// TIA Portal project "SPEEDGOAT_SimulaceSoustav_V20" (V20)

(* hardware
DEVICE "GSD device_1"  GSD.Device.PN
   slot 0: "Rack"  Rack  V1.0
   slot 0: "speedgoat-io750"  CIFX RE/PNS V3.4.19 - V3.4.x  1250.100  V3.4
      slot 0: "CIFX RE/PNS V3.4.19 - V3.4.x"  CIFX RE/PNS V3.4.19 - V3.4.x
      slot 1: "PN-IO"  PN-IO
         slot 1: "Port 1"  Port 1
         slot 2: "Port 2"  Port 2
   slot 1: "Model A - PN u"  4 Bytes Output
      slot 0: "4 Bytes Output"  4 Bytes Output
   slot 2: "Model A - PN y"  4 Bytes Input
      slot 0: "4 Bytes Input"  4 Bytes Input
DEVICE "S71500/ET200MP station_5"  S7-1500 station
   slot 0: "Rail_0"  Rack  6ES7 590-1***0-0AA0
   slot 1: "1500_ControlPLC"  CPU 1516-3 PN/DP  6ES7 516-3AN01-0AB0  V2.1
      slot 3: "CPU display_1"  6ES7591-1BA00-0AA0
   slot 2: "DI 32x24VDC HF_1"  DI 32x24VDC HF  6ES7 521-1BL00-0AB0  V2.0
   slot 3: "DQ 32x24VDC/0.5A HF_1"  DQ 32x24VDC/0.5A HF  6ES7 522-1BL01-0AB0  V1.0
   slot 4: "AQ 4xU/I ST_1"  AQ 4xU/I ST  6ES7 532-5HD00-0AB0  V2.0
   slot 5: "AI 8xU/I/RTD/TC ST_1"  AI 8xU/I/RTD/TC ST  6ES7 531-7KF00-0AB0  V2.0
DEVICE "GSD device_2"  GSD.Device.PN
   slot 0: "Rack"  Rack  V1.0
   slot 0: "speedgoat-io752"  CIFX RE/PNS V3.4.19 - V3.4.x  1250.100  V3.4
      slot 0: "CIFX RE/PNS V3.4.19 - V3.4.x"  CIFX RE/PNS V3.4.19 - V3.4.x
      slot 1: "PN-IO"  PN-IO
         slot 1: "Port 1"  Port 1
         slot 2: "Port 2"  Port 2
   slot 1: "Model C - PN u"  4 Bytes Output
      slot 0: "4 Bytes Output"  4 Bytes Output
   slot 2: "Model C - PN y"  4 Bytes Input
      slot 0: "4 Bytes Input"  4 Bytes Input
DEVICE "GSD device_3"  GSD.Device.PN
   slot 0: "Rack"  Rack  V1.0
   slot 0: "speedgoat-io751"  CIFX RE/PNS V3.4.19 - V3.4.x  1250.100  V3.4
      slot 0: "CIFX RE/PNS V3.4.19 - V3.4.x"  CIFX RE/PNS V3.4.19 - V3.4.x
      slot 1: "PN-IO"  PN-IO
         slot 1: "Port 1"  Port 1
         slot 2: "Port 2"  Port 2
   slot 1: "Model B - PN u"  4 Bytes Output
      slot 0: "4 Bytes Output"  4 Bytes Output
   slot 2: "Model B - PN y"  4 Bytes Input
      slot 0: "4 Bytes Input"  4 Bytes Input
DEVICE "HMI_1"  KTP900 Basic PN
   slot 0: "HMI_1"  KTP900 Basic PN  6AV2 123-2JB03-0AX0  15.1.0.0
   slot 1: "HMI_RT_1"  KTP900 Basic PN  6AV2 123-2JB03-0AX0  15.1.0.0
   slot 5: "HMI_1.IE_CP_1"  PROFINET Interface  15.0.1.0
      slot 1: "PROFINET Interface_1"  PROFINET Interface
         slot 1: "Port_1"  Port
DEVICE "GSD device_4"  GSD.Device.PN
   slot 0: "Rack"  Rack  V1.0
   slot 0: "speedgoat-io752_1"  CIFX RE/PNS V3.4.19 - V3.4.x  1250.100  V3.4
      slot 0: "CIFX RE/PNS V3.4.19 - V3.4.x"  CIFX RE/PNS V3.4.19 - V3.4.x
      slot 1: "PN-IO"  PN-IO
         slot 1: "Port 1"  Port 1
         slot 2: "Port 2"  Port 2
   slot 1: "Model C - PN u"  4 Bytes Output
      slot 0: "4 Bytes Output"  4 Bytes Output
   slot 2: "Model C - PN y"  4 Bytes Input
      slot 0: "4 Bytes Input"  4 Bytes Input
*)

// ===== PLC "1500_ControlPLC"  CPU 1516-3 PN/DP =====

VAR_GLOBAL   // PLC tag table "Process"
   "Only_Model_A_PN" AT %M20.0 : Bool;
   "Only_Model_B_PN" AT %M20.1 : Bool;
   "Only_Model_C_PN" AT %M20.2 : Bool;
   "SetPoint A" AT %MD54 : Real;
   "SetPoint B" AT %MD58 : Real;
   "SetPoint C" AT %MD62 : Real;
   "Model A - Reset" AT %M20.4 : Bool;
   "Model B - Reset" AT %M20.5 : Bool;
   "Model C - Reset" AT %M20.6 : Bool;
   "Connection_LOOPBACK" AT %M20.7 : Bool;   // Activates copying PROFINET input to output
   "Model A - PN u" AT %QD30 : Real;   // System A input (u) via PROFINET
   "Model B - PN u" AT %QD34 : Real;   // System B input (u) via PROFINET
   "Model C - PN u" AT %QD38 : Real;   // System C input (u) via PROFINET
   "Model A - PN y" AT %ID0 : Real;   // System A output (y) via PROFINET
   "Model B - PN y" AT %ID4 : Real;   // System B output (y) via PROFINET
   "Model C - PN y" AT %ID8 : Real;   // System C output (y) via PROFINET
   "Connection_PROFINET" AT %M20.3 : Bool;   // Activates closed loop control via PROFINET
   "Connection_LOCALMODEL" AT %M21.0 : Bool;   // Activates closed loop control with LOCAL MODELS
   "MEM 1" AT %M200.0 : Bool;   // E
   "MEM 2" AT %M200.1 : Bool;   // E
   "MEM 3" AT %M200.2 : Bool;   // E
   "MEM 4" AT %M200.3 : Bool;   // E
   "MEM 5" AT %M200.4 : Bool;   // E
   "MEM 6" AT %M200.5 : Bool;
   "MEM 7" AT %M200.6 : Bool;
   "MEM 8" AT %M200.7 : Bool;
   "MEM 9" AT %M201.0 : Bool;
   "MEM 10" AT %M201.1 : Bool;
   "MEM 11" AT %M201.2 : Bool;
   "MEM 12" AT %M201.3 : Bool;
   "MEM 13" AT %M201.4 : Bool;
   "MEM 14" AT %M201.5 : Bool;
   "MEM 15" AT %M201.6 : Bool;
   "MEM 16" AT %M201.7 : Bool;
   "MEM 17" AT %M202.0 : Bool;
   "MEM 18" AT %M202.1 : Bool;
   "Connection_NOCONNECTION" AT %M21.1 : Bool;
   "Connection_MANUALVALUE" AT %M21.2 : Bool;
   "resetModels" AT %M21.3 : Bool;
   "SetPoint D" AT %MD66 : Real;
   "Model D - PN u" AT %QD42 : Real;   // System D input (u) via PROFINET
   "Model D - PN y" AT %ID32 : Real;   // System D output (y) via PROFINET
   "EnablePID_D" AT %M21.4 : Bool;
   "SP DEMO" AT %M21.5 : Bool;
   "SP BINVAL" AT %M21.6 : Bool;
END_VAR

DATA_BLOCK "LSim_PDT1_DB"   // DB1
{ S7_Optimized_Access := 'TRUE' }
VERSION : 2.01
// stored: InstanceOfName LSim_PDT1
"LSim_PDT1"
BEGIN
END_DATA_BLOCK

DATA_BLOCK "Model_Params"   // DB2
{ S7_Optimized_Access := 'TRUE' }
VERSION : 0.1
   VAR
      "Model A" : Struct
         tmLag1 : Real := 3.0;
         tmLag2 : Real := 0.3;
         gain : Real := 1.25;
         cycle : Real := 0.2;
         maxOut : Real := 100.0;
         minOut : Real := 0.0;
      END_STRUCT;
      "Model B" : Struct
         tmLag1 : Real := 1.2;
         tmLag2 : Real := 0.25;
         gain : Real := 1.45;
         cycle : Real := 0.1;
         maxOut : Real := 100.0;
         minOut : Real := 0.0;
      END_STRUCT;
      "Model C" : Struct
         omega : Real := 2.0;
         damp : Real := 0.2;
         gain : Real := 1.33;
         cycle : Real := 0.05;
         maxOut : Real := 100.0;
         minOut : Real := 0.0;
      END_STRUCT;
   END_VAR
BEGIN
END_DATA_BLOCK

DATA_BLOCK "LSim_PT2aper_DB"   // DB3
{ S7_Optimized_Access := 'TRUE' }
VERSION : 2.01
// stored: InstanceOfName LSim_PT2aper
"LSim_PT2aper"
BEGIN
END_DATA_BLOCK

DATA_BLOCK "LSim_PT2osc_DB"   // DB8
{ S7_Optimized_Access := 'TRUE' }
VERSION : 2.01
// stored: InstanceOfName LSim_PT2osc
"LSim_PT2osc"
BEGIN
END_DATA_BLOCK

FUNCTION_BLOCK "LSim_PT2osc"   // FB52, SCL
{ S7_Optimized_Access := 'TRUE' }
VERSION : 2.01
   VAR_INPUT
      calcParam : Bool;   // recalculate with new parameters
      input : Real;   // input signal
      omega : Real := 2.0;   // angular frequency of the undampened vibrations [1/sec]
      damp : Real := 0.2;   // damping (0 < D < 1)
      gain : Real := 1.0;   // gain factor
      cycle : Real := 0.1;   // cyclic time [sec]
      maxOut : Real := 100.0;   // max. output limit
      minOut : Real;   // min. output limit
      reset : Bool;   // resets all relevant parameters to ‘0’ including the output
   END_VAR
   VAR_OUTPUT
      error : Bool;   // error (0 >= damp >= 1 or #omega <= 0)
      status : Word;   // status (if #error = TRUE then status = 16#8001)
      maxReached : Bool;   // output has reached max. limit
      minReached : Bool;   // output has reached min. limit
      output : Real;   // output signal (if #error = FALSE)
   END_VAR
   VAR
      statRxn2 : Real;   // delayed input signal (n-2)
      statRxn1 : Real;   // delayed input signal (n-1)
      statRyn2 : Real;   // delayed output signal (n-2)
      statRyn1 : Real;   // delayed output signal (n-1)
      statRb1 : Real;
      statRb2 : Real;
      statRa1 : Real;
      statRa2 : Real;
      statRo : Real;
      statSigma : Real;
      statNue : Real;
      statOverfirst : Bool;
      statOutput : Real;
   END_VAR
BEGIN
   //=============================================================================
   //SIEMENS AG
   //(c)Copyright 2017 All Rights Reserved
   //-----------------------------------------------------------------------------
   //Library:       Library for Controlled System Simulation
   //Tested with:   S7-1500 FW V2.0 / S7-1200 FW V4.2
   //Engineering:   STEP 7 V14 Upd2 (TIA Portal)
   //Restrictions:  Cyclic interrupt
   //Requirements:  memory card needed for S7-1500
   //Functionality: Simulation of a vibrating PT2-System
   //
   //                  gain
   //  F(p) = ----------------------------------
   //         SQR(p/omega) + 2*damp*p/omega + 1
   //          
   //  Call the simulation in a cyclic interrupt with
   //  cyclic interrupt time at least = tmLag1/10!
   //-----------------------------------------------------------------------------
   //Change log table:
   //Version  Date       Expert in charge                Changes applied
   //02.00.00 03.02.2016 Siemens Industry Online Support Release (STEP 7 V13 SP1)
   //02.00.01 02.03.2017 Siemens Industry Online Support Release (STEP 7 V14)
   //=============================================================================

   // check parameter
   IF #damp >= 1 OR #damp <= 0 OR #omega <= 0 THEN
     #error := TRUE;
     #status := W#16#8001;
     #statRxn1 := 0.0;
     #statRyn1 := 0.0;
     #statRxn2 := 0.0;
     #statRyn2 := 0.0;
     #statOutput := 0;
     #output := 0;
     RETURN;
   ELSE
     #error := FALSE;
     #status := W#16#0000;     // no error 
   END_IF;

   // calculates the z-parameter for the difference equatation
   IF #calcParam = True THEN
   // Calculate z-parameters for oscillating PT2-System
   #statRo := EXP(-2*#omega*#damp*#cycle);
   #statSigma := (COS(#omega * #cycle * SQRT(1 - SQR(#damp)))) * EXP(-#damp*#omega*#cycle);
   #statNue := (SIN(#omega*#cycle*SQRT(1-SQR(#damp)))) * (EXP(-#damp*#omega*#cycle)) * (#damp / SQRT(1 - SQR(#damp)));
   #statRa1 := -2*#statSigma;
   #statRa2 := #statRo;
   #statRb1 := #gain*(1 - #statSigma - #statNue);
   #statRb2 := #gain*(#statRo - #statSigma + #statNue);
   END_IF;

   // reset Memory
   IF #reset = True THEN
     #statRxn1 := 0.0;
     #statRyn1 := 0.0;
     #statRxn2 := 0.0;
     #statRyn2 := 0.0;
     #statOutput:=0;
     #error := False;
     #status := W#16#0000;
   END_IF;

   // save delayed output signals
   #statRyn2:=#statRyn1;
   #statRyn1:= #statOutput;

   // difference equatation for PT2-System
   #statOutput := #statRxn1* #statRb1 + #statRxn2*#statRb2 - #statRyn1*#statRa1 - #statRyn2*#statRa2;

   // save delayed input signals
   #statRxn2 := #statRxn1;
   #statRxn1 := #input;

   // max limit of acutating variable
   IF #statOutput > #maxOut THEN
     #statOutput := #maxOut;
     #maxReached:= True;
   ELSE
     #maxReached := False;
   END_IF;

   // min limit of acutating variable
   IF #statOutput < #minOut THEN
     #statOutput := #minOut;
     #minReached := True;
   ELSE
     #minReached := False;
   END_IF;

   #output := #statOutput;
END_FUNCTION_BLOCK

FUNCTION_BLOCK "LSim_PT2aper"   // FB53, SCL
{ S7_Optimized_Access := 'TRUE' }
VERSION : 2.01
   VAR_INPUT
      calcParam : Bool;   // recalculate with new parameters
      input : Real;   // input signal
      tmLag1 : Real := 2.0;   // time constant T1 [sec]
      tmLag2 : Real := 0.2;   // time constant T2 [sec]
      gain : Real := 1.0;   // gain factor
      cycle : Real := 0.1;   // cyclic time [sec]
      maxOut : Real := 100.0;   // max. output limit
      minOut : Real;   // min. output limit
      reset : Bool;   // resets all relevant parameters to ‘0’ including the output
   END_VAR
   VAR_OUTPUT
      error : Bool;   // error (#tmLag1 <= 0 or #tmLag2 <= 0 or #tmLag1 = #tmLag2)
      status : Word;   // status (if #error = TRUE then status = 16#8001)
      maxReached : Bool;   // output has reached max. limit
      minReached : Bool;   // output has reached min. limit
      output : Real;   // output signal (if #error = FALSE)
   END_VAR
   VAR
      statRxn2 : Real;   // delayed input signal (n-2)
      statRxn1 : Real;   // delayed input signal (n-1)
      statRyn2 : Real;   // delayed output signal (n-2)
      statRyn1 : Real;   // delayed output signal (n-1)
      statRf1 : Real;
      statRf2 : Real;
      statRe1 : Real;
      statRe2 : Real;
      statAlpha : Real;
      statBeta : Real;
      statGamma : Real;
      statDelta : Real;
      statOverfirst : Bool;
      statOutput : Real;   // Output signal
   END_VAR
BEGIN
   //=============================================================================
   //SIEMENS AG
   //(c)Copyright 2017 All Rights Reserved
   //-----------------------------------------------------------------------------
   //Library:       Library for Controlled System Simulation
   //Tested with:   S7-1500 FW V2.0 / S7-1200 FW V4.2
   //Engineering:   STEP 7 V14 Upd2 (TIA Portal)
   //Restrictions:  Cyclic interrupt
   //Requirements:  memory card needed for S7-1500
   //Functionality: Simulation of a aperiodic PT2-System
   //  
   //                    gain
   //  F(p) = -----------------------------
   //         (tmLag1*p + 1)*(tmLag2*p + 1)
   //         
   //  Call the simulation in a cyclic interrupt with
   //  cyclic interrupt time at least = tmLag1/10!
   //-----------------------------------------------------------------------------
   //Change log table:
   //Version  Date       Expert in charge                Changes applied
   //02.00.00 03.02.2016 Siemens Industry Online Support Release (STEP 7 V13 SP1)
   //02.00.01 02.03.2017 Siemens Industry Online Support Release (STEP 7 V14)
   //=============================================================================

   // check parameter
   IF #tmLag1 <= 0 OR #tmLag2 <= 0 OR #tmLag1 = #tmLag2 THEN
     #error := TRUE;
     #status := W#16#8001;     // Parameter Error
     #statRxn1 := 0.0;
     #statRyn1 := 0.0;
     #statRxn2 := 0.0;
     #statRyn2 := 0.0;
     #statOutput := 0;
     #output := 0;
     RETURN;
   ELSE
     #error := FALSE;
     #status := W#16#0000;     // no error
   END_IF;

   // calculates the z-parameter for the difference equatation
   IF #calcParam = True OR NOT #statOverfirst THEN
     #statOverfirst := 1;
     // Calculate z-parameters for IT1-System
     #statAlpha := EXP(- #cycle / #tmLag1);
     #statBeta := EXP(- #cycle / #tmLag2);
     #statGamma := #tmLag1 / (#tmLag1 - #tmLag2);
     #statDelta := #tmLag2 / (#tmLag1 - #tmLag2);
     #statRe1 := - #statAlpha - #statBeta;
     #statRe2 := #statAlpha * #statBeta;
     #statRf1 := #gain * (1 - #statGamma * #statAlpha + #statDelta * #statBeta);
     #statRf2 := #gain * (#statAlpha * #statBeta - #statGamma * #statBeta + #statAlpha * #statDelta);
   END_IF;

   // reset Memory
   IF #reset = True THEN
     #statRxn1 := 0.0;
     #statRyn1 := 0.0;
     #statRxn2 := 0.0;
     #statRyn2 := 0.0;
     #statOutput := 0;
   END_IF;
   //save delayed input signals
   #statRxn2 := #statRxn1;
   #statRxn1 := #input;

   //save delayed output signals
   #statRyn2:=#statRyn1;
   #statRyn1:= #statOutput;

   // difference equatation of the PT2-System
   #statOutput := #statRxn1* #statRf1 + #statRxn2*#statRf2 - #statRyn1*#statRe1 - #statRyn2*#statRe2;

   // max limit of acutating variable
   IF #statOutput > #maxOut THEN
     #statOutput := #maxOut;
     #maxReached:= True;
   ELSE
     #maxReached := False;
   END_IF;

   // min limit of acutating variable
   IF #statOutput < #minOut THEN
     #statOutput := #minOut;
     #minReached := True;
   ELSE
     #minReached := False;
   END_IF;

   #output := #statOutput;
END_FUNCTION_BLOCK

FUNCTION_BLOCK "LSim_PDT1"   // FB55, SCL
{ S7_Optimized_Access := 'TRUE' }
VERSION : 2.01
   VAR_INPUT
      calcParam : Bool;   // recalculate with new parameters
      input : Real;   // input signal
      tmLag1 : Real := 2.0;   // time constant T1 [sec]
      tmLag2 : Real := 0.2;   // time constant T2 [sec]
      gain : Real := 1.0;   // gain factor
      cycle : Real := 0.1;   // cyclic time [sec]
      maxOut : Real := 100.0;   // max. output limit
      minOut : Real;   // min. output limit
      reset : Bool;   // resets all relevant parameters to ‘0’ including the output
   END_VAR
   VAR_OUTPUT
      error : Bool;   // error (#tmLag1 <= 0 or #tmLag2 <= 0)
      status : Word;   // status (if #error = TRUE then status = 16#8001)
      maxReached : Bool;   // output has reached max. limit
      minReached : Bool;   // output has reached min. limit
      output : Real;   // output signal (if #error = FALSE)
   END_VAR
   VAR
      statRxn2 : Real;   // delayed input signal (n-2)
      statRxn1 : Real;   // delayed input signal (n-1)
      statRyn2 : Real;   // delayed output signal (n-2)
      statRyn1 : Real;   // delayed output signal (n-1)
      statRb1 : Real;
      statRb0 : Real;
      statRa1 : Real;
      statOverfirst : Bool;
      statOutput : Real;
   END_VAR
BEGIN
   //=============================================================================
   //SIEMENS AG
   //(c)Copyright 2017 All Rights Reserved
   //-----------------------------------------------------------------------------
   //Library:       Library for Controlled System Simulation
   //Tested with:   S7-1500 FW V2.0 / S7-1200 FW V4.2
   //Engineering:   STEP 7 V14 Upd2 (TIA Portal)
   //Restrictions:  Cyclic interrupt
   //Requirements:  memory card needed for S7-1500
   //Functionality: Simulation of an PD-T1 System
   //
   //         gain * (1 + tmLag2*p)
   //  F(p) = ------------------------------
   //            (1 + tmLag1*p)
   //          
   //  Call the simulation in a cyclic interrupt with
   //  cyclic interrupt time at least = tmLag1/10!
   //-----------------------------------------------------------------------------
   //Change log table:
   //Version  Date       Expert in charge                Changes applied
   //02.00.00 03.02.2016 Siemens Industry Online Support Release (STEP 7 V13 SP1)
   //02.00.01 02.03.2017 Siemens Industry Online Support Release (STEP 7 V14)
   //=============================================================================

   // check parameter
   IF #tmLag1 <= 0 OR #tmLag2 <= 0 THEN
     #error := True;
     #status := W#16#8001;     // Parameter Error
     #statRxn1 := 0.0;
     #statRyn1 := 0.0;
     #statRxn2 := 0.0;
     #statRyn2 := 0.0;
     #statOutput := 0;
     #output := 0;
     RETURN;
   ELSE
     #error := FALSE;
     #status := W#16#0000;     // no error
   END_IF;

   // calculates the z-parameter for the difference equatation
   IF #calcParam = True OR NOT #statOverfirst THEN
     #statOverfirst := 1;
   // Calculate z-parameters for oscilating PT2-System
   #statRa1 := -EXP(-#cycle/#tmLag1);
   #statRb0 := #gain *(#tmLag2/#tmLag1);
   #statRb1 := #gain *(1 + #statRa1 - (#tmLag2/#tmLag1));
   END_IF;

   // reset Memory
   IF #reset = True THEN
     #statRxn1 := 0.0;
     #statRyn1 := 0.0;
     #statRxn2 := 0.0;
     #statRyn2 := 0.0;
     #statOutput:=0;
     #error := False;
     #status := W#16#0000;
   END_IF;

   // save delayed output-signals
   #statRyn1:= #statOutput;

   // difference equatation for PT2-system
   #statOutput := #input * #statRb0 +  #statRxn1* #statRb1 - #statRyn1*#statRa1;

   // save delayed input-signals
   #statRxn1 := #input;

   // max limit of acutating variable
   IF #statOutput > #maxOut THEN
     #statOutput := #maxOut;
     #maxReached:= True;
   ELSE
     #maxReached := False;
   END_IF;

   // min limit of acutating variable
   IF #statOutput < #minOut THEN
     #statOutput := #minOut;
     #minReached := True;
   ELSE
     #minReached := False;
   END_IF;

   #output := #statOutput;
END_FUNCTION_BLOCK

FUNCTION "ConnectionSwitch" : Void   // FC1, SCL
{ S7_Optimized_Access := 'TRUE' }
VERSION : 0.1
   VAR CONSTANT
      "Default value" : Real := 0.0;
   END_VAR
BEGIN
   IF "Connection_LOCALMODEL" THEN
       // Model A from local instance
       "PID_Compact_Control_A".Input := "LSim_PDT1_DB".output;
       "LSim_PDT1_DB".input := "PID_Compact_Control_A".Output;
       // Model B from local instance
       "PID_Compact_Control_B".Input := "LSim_PT2aper_DB".output;
       "LSim_PT2aper_DB".input := "PID_Compact_Control_B".Output;
       // Model C from local instance
       "PID_Compact_Control_C".Input := "LSim_PT2osc_DB".output;
       "LSim_PT2osc_DB".input := "PID_Compact_Control_C".Output;
       // Model D - nothing
       IF "EnablePID_D" = TRUE THEN
           "EnablePID_D" := FALSE;
       END_IF;

   ELSIF "Connection_PROFINET" THEN
       "EnablePID_D" := TRUE;
       // Model A from PN
       "PID_Compact_Control_A".Input := "Model A - PN y";
       "Model A - PN u" := "PID_Compact_Control_A".Output;
       // Model B from PN
       "PID_Compact_Control_B".Input := "Model B - PN y";
       "Model B - PN u" := "PID_Compact_Control_B".Output;
       // Model C from PN
       "PID_Compact_Control_C".Input := "Model C - PN y";
       "Model C - PN u" := "PID_Compact_Control_C".Output;
       // Model D fron PN
       "PID_Compact_Control_D".Input := "Model D - PN y";
       "Model D - PN u" := "PID_Compact_Control_D".Output;
   ELSIF "Connection_LOOPBACK" THEN
       "Model A - PN u" := "Model A - PN y";
       "Model B - PN u" := "Model B - PN y";
       "Model C - PN u" := "Model C - PN y";
       "Model D - PN u" := "Model D - PN y";
   ELSIF "Connection_MANUALVALUE" THEN
       "Model A - PN u" := "SetPoint A";
       "Model B - PN u" := "SetPoint B";
       "Model C - PN u" := "SetPoint C";
       "Model D - PN u" := "SetPoint D";
       IF "EnablePID_D" = TRUE THEN
           "EnablePID_D" := FALSE;
       END_IF;
   ELSE
       "Model A - PN u" := #"Default value";
       "Model B - PN u" := #"Default value";
       "Model C - PN u" := #"Default value";
       "Model D - PN u" := #"Default value";
       IF "EnablePID_D" = TRUE THEN
           "EnablePID_D" := FALSE;
       END_IF;
   END_IF;
END_FUNCTION

ORGANIZATION_BLOCK "Main"   // OB1, LAD, ProgramCycle
TITLE = "Main Program Sweep (Cycle)"
{ S7_Optimized_Access := 'TRUE' }
VERSION : 0.1
   VAR_INPUT
      Initial_Call : Bool;   // Initial call of this OB
      Remanence : Bool;   // =True, if remanent data are available
   END_VAR
   VAR_TEMP   // added for the SCL form of the ladder/FBD networks
      _w1 : Bool;
      _w2 : Bool;
      _w3 : Bool;
      _w4 : Bool;
      _w5 : Bool;
      _w6 : Bool;
   END_VAR
BEGIN

REGION Network 1: Connection switch
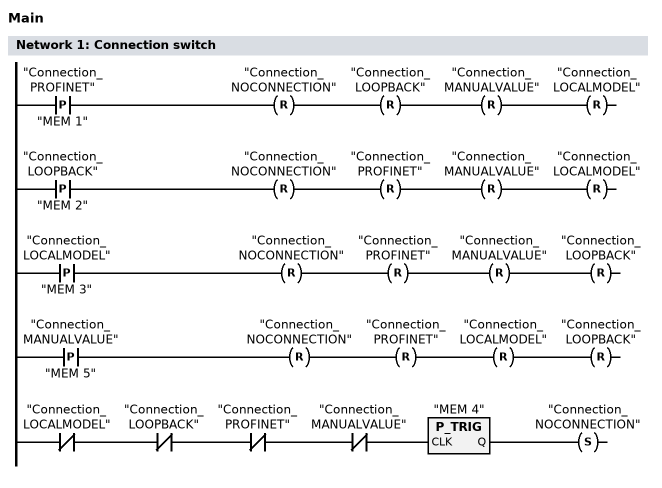
   RUNG wire#powerrail
      P_Contact(operand := "Connection_PROFINET", bit := "MEM 1")
      R_Coil( "Connection_NOCONNECTION" )
      R_Coil( "Connection_LOOPBACK" )
      R_Coil( "Connection_MANUALVALUE" )
      R_Coil( "Connection_LOCALMODEL" )
   END_RUNG
   RUNG wire#powerrail
      P_Contact(operand := "Connection_LOOPBACK", bit := "MEM 2")
      R_Coil( "Connection_NOCONNECTION" )
      R_Coil( "Connection_PROFINET" )
      R_Coil( "Connection_MANUALVALUE" )
      R_Coil( "Connection_LOCALMODEL" )
   END_RUNG
   RUNG wire#powerrail
      P_Contact(operand := "Connection_LOCALMODEL", bit := "MEM 3")
      R_Coil( "Connection_NOCONNECTION" )
      R_Coil( "Connection_PROFINET" )
      R_Coil( "Connection_MANUALVALUE" )
      R_Coil( "Connection_LOOPBACK" )
   END_RUNG
   RUNG wire#powerrail
      P_Contact(operand := "Connection_MANUALVALUE", bit := "MEM 5")
      R_Coil( "Connection_NOCONNECTION" )
      R_Coil( "Connection_PROFINET" )
      R_Coil( "Connection_LOCALMODEL" )
      R_Coil( "Connection_LOOPBACK" )
   END_RUNG
   RUNG wire#powerrail
      I_Contact( "Connection_LOCALMODEL" )
      I_Contact( "Connection_LOOPBACK" )
      I_Contact( "Connection_PROFINET" )
      I_Contact( "Connection_MANUALVALUE" )
      P_Trig( "MEM 4" )
      S_Coil( "Connection_NOCONNECTION" )
   END_RUNG
   // the same network as SCL:
   #_w1 := "Connection_PROFINET" AND NOT "MEM 1";   // rising edge of "Connection_PROFINET"
   "MEM 1" := "Connection_PROFINET";
   IF #_w1 THEN
       "Connection_NOCONNECTION" := FALSE;
       "Connection_LOOPBACK" := FALSE;
       "Connection_MANUALVALUE" := FALSE;
       "Connection_LOCALMODEL" := FALSE;
   END_IF;
   #_w2 := "Connection_LOOPBACK" AND NOT "MEM 2";   // rising edge of "Connection_LOOPBACK"
   "MEM 2" := "Connection_LOOPBACK";
   IF #_w2 THEN
       "Connection_NOCONNECTION" := FALSE;
       "Connection_PROFINET" := FALSE;
       "Connection_MANUALVALUE" := FALSE;
       "Connection_LOCALMODEL" := FALSE;
   END_IF;
   #_w3 := "Connection_LOCALMODEL" AND NOT "MEM 3";   // rising edge of "Connection_LOCALMODEL"
   "MEM 3" := "Connection_LOCALMODEL";
   IF #_w3 THEN
       "Connection_NOCONNECTION" := FALSE;
       "Connection_PROFINET" := FALSE;
       "Connection_MANUALVALUE" := FALSE;
       "Connection_LOOPBACK" := FALSE;
   END_IF;
   #_w4 := "Connection_MANUALVALUE" AND NOT "MEM 5";   // rising edge of "Connection_MANUALVALUE"
   "MEM 5" := "Connection_MANUALVALUE";
   IF #_w4 THEN
       "Connection_NOCONNECTION" := FALSE;
       "Connection_PROFINET" := FALSE;
       "Connection_LOCALMODEL" := FALSE;
       "Connection_LOOPBACK" := FALSE;
   END_IF;
   #_w5 := NOT "Connection_LOCALMODEL" AND NOT "Connection_LOOPBACK" AND NOT "Connection_PROFINET" AND NOT "Connection_MANUALVALUE";
   #_w6 := #_w5 AND NOT "MEM 4";   // rising edge
   "MEM 4" := #_w5;
   IF #_w6 THEN "Connection_NOCONNECTION" := TRUE; END_IF;
END_REGION
END_ORGANIZATION_BLOCK

ORGANIZATION_BLOCK "Control A"   // OB30, LAD, CyclicInterrupt
TITLE = Simulation and control of an PD-T1 System
{ S7_Optimized_Access := 'TRUE' }
VERSION : 0.1
   VAR_INPUT
      Initial_Call : Bool;   // Initial call of this OB
      Event_Count : Int;   // Events discarded
   END_VAR
BEGIN

REGION Network 1: Model of PDT1
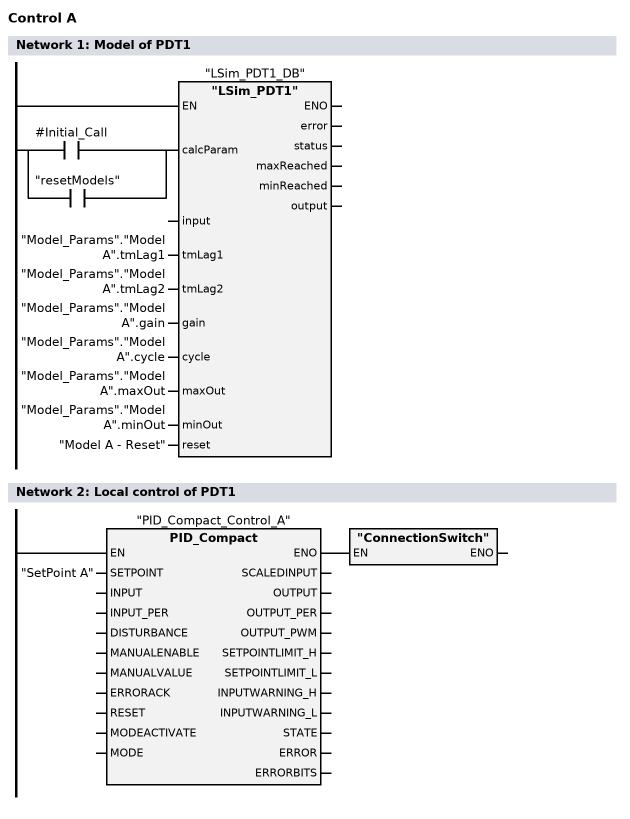
   RUNG wire#powerrail
      "LSim_PDT1_DB"(calcParam := wire#w1, input :=, tmLag1 := "Model_Params"."Model A".tmLag1, tmLag2 := "Model_Params"."Model A".tmLag2, gain := "Model_Params"."Model A".gain, cycle := "Model_Params"."Model A".cycle, maxOut := "Model_Params"."Model A".maxOut, minOut := "Model_Params"."Model A".minOut, reset := "Model A - Reset", error =>, status =>, maxReached =>, minReached =>, output =>)
   END_RUNG
   RUNG wire#powerrail
      Contact( #Initial_Call )
   END_RUNG wire#w1
   RUNG wire#powerrail
      Contact( "resetModels" )
   END_RUNG wire#w1
   // the same network as SCL:
   "LSim_PDT1_DB"(calcParam := #Initial_Call OR "resetModels",   // "LSim_PDT1"
                  tmLag1 := "Model_Params"."Model A".tmLag1,
                  tmLag2 := "Model_Params"."Model A".tmLag2,
                  gain := "Model_Params"."Model A".gain,
                  cycle := "Model_Params"."Model A".cycle,
                  maxOut := "Model_Params"."Model A".maxOut,
                  minOut := "Model_Params"."Model A".minOut,
                  reset := "Model A - Reset");
END_REGION

REGION Network 2: Local control of PDT1
   // ENO of a box is taken as its EN; it also drops when the box reports an error
   "PID_Compact_Control_A"(Setpoint := "SetPoint A");   // PID_Compact
   "ConnectionSwitch"();
END_REGION

REGION Network 3: Connection switch
END_REGION
END_ORGANIZATION_BLOCK

ORGANIZATION_BLOCK "Control B"   // OB31, LAD, CyclicInterrupt
TITLE = Simulation and control of an PT2aper system
{ S7_Optimized_Access := 'TRUE' }
VERSION : 0.1
   VAR_INPUT
      Initial_Call : Bool;   // Initial call of this OB
      Event_Count : Int;   // Events discarded
   END_VAR
BEGIN

REGION Network 1: Model of PT2aper
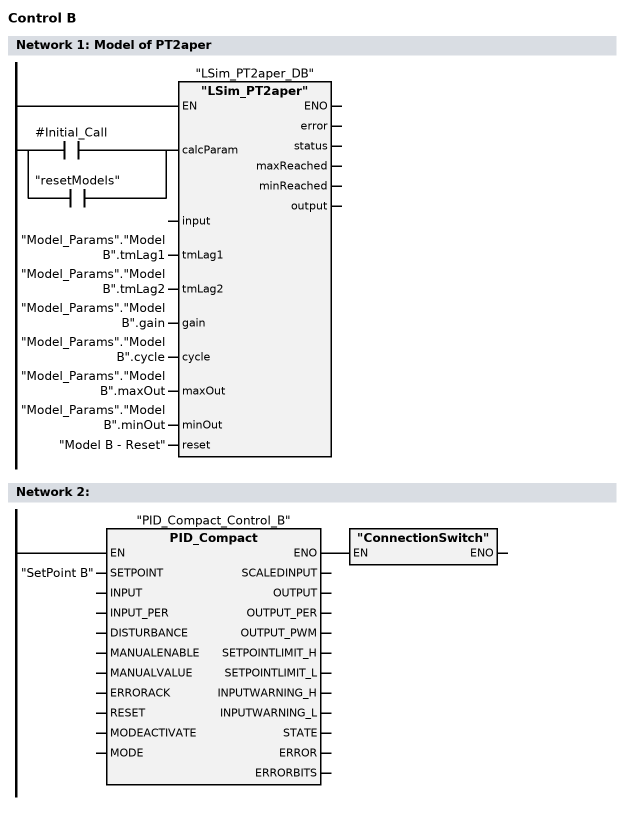
   RUNG wire#powerrail
      "LSim_PT2aper_DB"(calcParam := wire#w1, input :=, tmLag1 := "Model_Params"."Model B".tmLag1, tmLag2 := "Model_Params"."Model B".tmLag2, gain := "Model_Params"."Model B".gain, cycle := "Model_Params"."Model B".cycle, maxOut := "Model_Params"."Model B".maxOut, minOut := "Model_Params"."Model B".minOut, reset := "Model B - Reset", error =>, status =>, maxReached =>, minReached =>, output =>)
   END_RUNG
   RUNG wire#powerrail
      Contact( #Initial_Call )
   END_RUNG wire#w1
   RUNG wire#powerrail
      Contact( "resetModels" )
   END_RUNG wire#w1
   // the same network as SCL:
   "LSim_PT2aper_DB"(calcParam := #Initial_Call OR "resetModels",   // "LSim_PT2aper"
                     tmLag1 := "Model_Params"."Model B".tmLag1,
                     tmLag2 := "Model_Params"."Model B".tmLag2,
                     gain := "Model_Params"."Model B".gain,
                     cycle := "Model_Params"."Model B".cycle,
                     maxOut := "Model_Params"."Model B".maxOut,
                     minOut := "Model_Params"."Model B".minOut,
                     reset := "Model B - Reset");
END_REGION

REGION Network 2
   // ENO of a box is taken as its EN; it also drops when the box reports an error
   "PID_Compact_Control_B"(Setpoint := "SetPoint B");   // PID_Compact
   "ConnectionSwitch"();
END_REGION
END_ORGANIZATION_BLOCK

ORGANIZATION_BLOCK "Control C"   // OB32, LAD, CyclicInterrupt
TITLE = Simulation and control of an PT3 system
{ S7_Optimized_Access := 'TRUE' }
VERSION : 0.1
   VAR_INPUT
      Initial_Call : Bool;   // Initial call of this OB
      Event_Count : Int;   // Events discarded
   END_VAR
BEGIN

REGION Network 1: Model of PT3 system
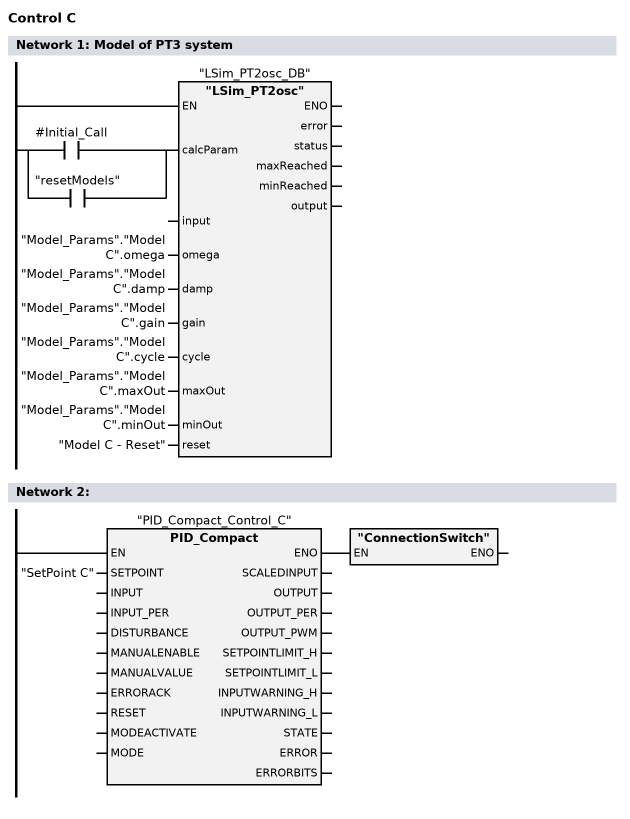
   RUNG wire#powerrail
      "LSim_PT2osc_DB"(calcParam := wire#w1, input :=, omega := "Model_Params"."Model C".omega, damp := "Model_Params"."Model C".damp, gain := "Model_Params"."Model C".gain, cycle := "Model_Params"."Model C".cycle, maxOut := "Model_Params"."Model C".maxOut, minOut := "Model_Params"."Model C".minOut, reset := "Model C - Reset", error =>, status =>, maxReached =>, minReached =>, output =>)
   END_RUNG
   RUNG wire#powerrail
      Contact( #Initial_Call )
   END_RUNG wire#w1
   RUNG wire#powerrail
      Contact( "resetModels" )
   END_RUNG wire#w1
   // the same network as SCL:
   "LSim_PT2osc_DB"(calcParam := #Initial_Call OR "resetModels",   // "LSim_PT2osc"
                    omega := "Model_Params"."Model C".omega,
                    damp := "Model_Params"."Model C".damp,
                    gain := "Model_Params"."Model C".gain,
                    cycle := "Model_Params"."Model C".cycle,
                    maxOut := "Model_Params"."Model C".maxOut,
                    minOut := "Model_Params"."Model C".minOut,
                    reset := "Model C - Reset");
END_REGION

REGION Network 2
   // ENO of a box is taken as its EN; it also drops when the box reports an error
   "PID_Compact_Control_C"(Setpoint := "SetPoint C");   // PID_Compact
   "ConnectionSwitch"();
END_REGION
END_ORGANIZATION_BLOCK

ORGANIZATION_BLOCK "Control D - FastTest"   // OB33, LAD, CyclicInterrupt
{ S7_Optimized_Access := 'TRUE' }
VERSION : 0.1
   VAR_INPUT
      Initial_Call : Bool;   // Initial call of this OB
      Event_Count : Int;   // Events discarded
   END_VAR
   VAR_TEMP   // added for the SCL form of the ladder/FBD networks
      _w1 : Bool;
   END_VAR
BEGIN

REGION Network 1
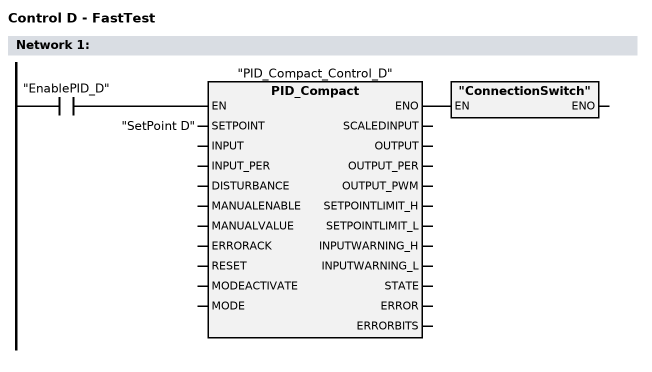
   // ENO of a box is taken as its EN; it also drops when the box reports an error
   #_w1 := "EnablePID_D";
   IF #_w1 THEN
       "PID_Compact_Control_D"(Setpoint := "SetPoint D");   // PID_Compact
       "ConnectionSwitch"();
   END_IF;
END_REGION
END_ORGANIZATION_BLOCK

ORGANIZATION_BLOCK "DEMO Setpoint"   // OB34, LAD, CyclicInterrupt
{ S7_Optimized_Access := 'TRUE' }
VERSION : 0.1
   VAR_INPUT
      Initial_Call : Bool;   // Initial call of this OB
      Event_Count : Int;   // Events discarded
   END_VAR
   VAR_TEMP   // added for the SCL form of the ladder/FBD networks
      _w1 : Bool;
      _w2 : Bool;
   END_VAR
BEGIN

REGION Network 1
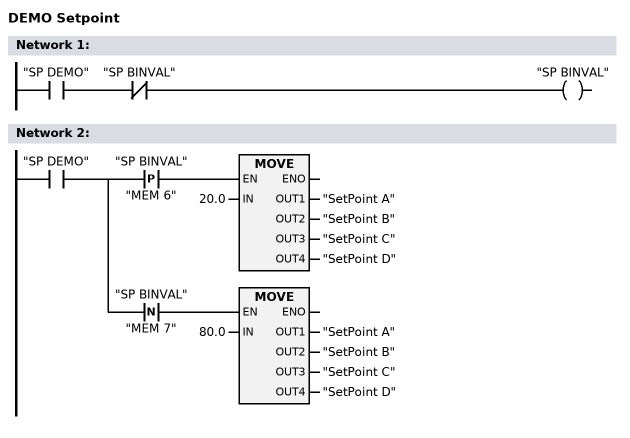
   RUNG wire#powerrail
      Contact( "SP DEMO" )
      I_Contact( "SP BINVAL" )
      Coil( "SP BINVAL" )
   END_RUNG
   // the same network as SCL:
   "SP BINVAL" := "SP DEMO" AND NOT "SP BINVAL";
END_REGION

REGION Network 2
   RUNG wire#powerrail
      Contact( "SP DEMO" )
      wire#w1
      P_Contact(operand := "SP BINVAL", bit := "MEM 6")
      Move(in := 20.0, out1 => "SetPoint A", out2 => "SetPoint B", out3 => "SetPoint C", out4 => "SetPoint D")
   END_RUNG
   RUNG wire#w1
      N_Contact(operand := "SP BINVAL", bit := "MEM 7")
      Move(in := 80.0, out1 => "SetPoint A", out2 => "SetPoint B", out3 => "SetPoint C", out4 => "SetPoint D")
   END_RUNG
   // the same network as SCL:
   #_w1 := "SP DEMO" AND "SP BINVAL" AND NOT "MEM 6";   // rising edge of "SP BINVAL"
   "MEM 6" := "SP BINVAL";
   IF #_w1 THEN
       "SetPoint A" := 20.0;
       "SetPoint B" := 20.0;
       "SetPoint C" := 20.0;
       "SetPoint D" := 20.0;
   END_IF;
   #_w2 := "SP DEMO" AND NOT "SP BINVAL" AND "MEM 7";   // falling edge of "SP BINVAL"
   "MEM 7" := "SP BINVAL";
   IF #_w2 THEN
       "SetPoint A" := 80.0;
       "SetPoint B" := 80.0;
       "SetPoint C" := 80.0;
       "SetPoint D" := 80.0;
   END_IF;
END_REGION
END_ORGANIZATION_BLOCK

ORGANIZATION_BLOCK "Startup"   // OB100, SCL, Startup
TITLE = "Complete Restart"
{ S7_Optimized_Access := 'TRUE' }
VERSION : 0.1
   VAR_INPUT
      LostRetentive : Bool;   // True if retentive data are lost
      LostRTC : Bool;   // True if date and time are lost
   END_VAR
BEGIN
   "Connection_LOCALMODEL" := 0;
   "Connection_LOOPBACK" := 0;
   "Connection_PROFINET" := 0;
   "Connection_MANUALVALUE" := 0;
   "Connection_NOCONNECTION" := 1;
END_ORGANIZATION_BLOCK

(* ===== HMI "HMI_RT_1" =====
system functions are stored by id; their names below are inferred from use
connection "HMI_Connection_1": ETHERNET, SMART_S7_1500_OMS

HMI tags "Default tag table"
   "Tag_ScreenNumber" : UInt, internal
   "Connection_PROFINET" : Bool = PLC Connection_PROFINET AT %M20.3, 1 s
   "Connection_LOOPBACK" : Bool = PLC Connection_LOOPBACK AT %M20.7, 1 s
   "Connection_LOCALMODEL" : Bool = PLC Connection_LOCALMODEL AT %M21.0, 1 s
   "Connection_NOCONNECTION" : Bool = PLC Connection_NOCONNECTION AT %M21.1, 1 s
   "Connection_LOCALVALUE" : Bool = PLC Connection_MANUALVALUE AT %M21.2, 1 s
   "PID_Compact_Control_A_Input" : Real = PLC PID_Compact_Control_A.Input, 1 s
   "PID_Compact_Control_B_Input" : Real = PLC PID_Compact_Control_B.Input, 1 s
   "PID_Compact_Control_C_Input" : Real = PLC PID_Compact_Control_C.Input, 1 s
   "PID_Compact_Control_A_Output" : Real = PLC PID_Compact_Control_A.Output, 1 s
   "PID_Compact_Control_B_Output" : Real = PLC PID_Compact_Control_B.Output, 1 s
   "PID_Compact_Control_C_Output" : Real = PLC PID_Compact_Control_C.Output, 1 s
   "LSim_PDT1_DB_input" : Real = PLC LSim_PDT1_DB.input, 1 s
   "LSim_PT2aper_DB_input" : Real = PLC LSim_PT2aper_DB.input, 1 s
   "LSim_PDT1_DB_output" : Real = PLC LSim_PDT1_DB.output, 1 s
   "LSim_PT2aper_DB_output" : Real = PLC LSim_PT2aper_DB.output, 1 s
   "Model A - PN u" : Real = PLC "Model A - PN u" AT %QD30, 1 s
   "Model B - PN u" : Real = PLC "Model B - PN u" AT %QD34, 1 s
   "Model C - PN u" : Real = PLC "Model C - PN u" AT %QD38, 1 s
   "Model A - PN y" : Real = PLC "Model A - PN y" AT %ID0, 1 s
   "Model B - PN y" : Real = PLC "Model B - PN y" AT %ID4, 1 s
   "Model C - PN y" : Real = PLC "Model C - PN y" AT %ID8, 1 s
   "SetPoint A" : Real = PLC "SetPoint A" AT %MD54, 1 s
   "SetPoint B" : Real = PLC "SetPoint B" AT %MD58, 1 s
   "SetPoint C" : Real = PLC "SetPoint C" AT %MD62, 1 s
   "LSim_PT2osc_DB_input" : Real = PLC LSim_PT2osc_DB.input, 1 s
   "LSim_PT2osc_DB_output" : Real = PLC LSim_PT2osc_DB.output, 1 s
   "PID_Compact_Control_A_Retain_CtrlParams_Gain" : Real = PLC PID_Compact_Control_A.Retain.CtrlParams.Gain, 1 s
   "PID_Compact_Control_A_Retain_CtrlParams_Ti" : Real = PLC PID_Compact_Control_A.Retain.CtrlParams.Ti, 1 s
   "PID_Compact_Control_A_Retain_CtrlParams_Td" : Real = PLC PID_Compact_Control_A.Retain.CtrlParams.Td, 1 s
   "PID_Compact_Control_B_Retain_CtrlParams_Gain" : Real = PLC PID_Compact_Control_B.Retain.CtrlParams.Gain, 1 s
   "PID_Compact_Control_B_Retain_CtrlParams_Ti" : Real = PLC PID_Compact_Control_B.Retain.CtrlParams.Ti, 1 s
   "PID_Compact_Control_B_Retain_CtrlParams_Td" : Real = PLC PID_Compact_Control_B.Retain.CtrlParams.Td, 1 s
   "PID_Compact_Control_C_Retain_CtrlParams_Gain" : Real = PLC PID_Compact_Control_C.Retain.CtrlParams.Gain, 1 s
   "PID_Compact_Control_C_Retain_CtrlParams_Ti" : Real = PLC PID_Compact_Control_C.Retain.CtrlParams.Ti, 1 s
   "PID_Compact_Control_C_Retain_CtrlParams_Td" : Real = PLC PID_Compact_Control_C.Retain.CtrlParams.Td, 1 s
   "PID_Compact_Control_A_Retain_CtrlParams_Cycle" : Real = PLC PID_Compact_Control_A.Retain.CtrlParams.Cycle, 1 s
   "PID_Compact_Control_B_Retain_CtrlParams_Cycle" : Real = PLC PID_Compact_Control_B.Retain.CtrlParams.Cycle, 1 s
   "PID_Compact_Control_C_Retain_CtrlParams_Cycle" : Real = PLC PID_Compact_Control_C.Retain.CtrlParams.Cycle, 1 s
   "PID_Compact_Control_D_CycleTime_Value" : Real = PLC PID_Compact_Control_D.CycleTime.Value, 1 s
   "SetPoint D" : Real = PLC "SetPoint D" AT %MD66, 1 s
   "PID_Compact_Control_D_Retain_CtrlParams_Gain" : Real = PLC PID_Compact_Control_D.Retain.CtrlParams.Gain, 1 s
   "PID_Compact_Control_D_Retain_CtrlParams_Ti" : Real = PLC PID_Compact_Control_D.Retain.CtrlParams.Ti, 1 s
   "PID_Compact_Control_D_Retain_CtrlParams_Td" : Real = PLC PID_Compact_Control_D.Retain.CtrlParams.Td, 1 s
   "PID_Compact_Control_D_Retain_CtrlParams_Cycle" : Real = PLC PID_Compact_Control_D.Retain.CtrlParams.Cycle, 1 s
   "Model D - PN u" : Real = PLC "Model D - PN u" AT %QD42, 1 s
   "Model D - PN y" : Real = PLC "Model D - PN y" AT %ID32, 1 s

text list "Btn_ConnectionMode": 0 'Activate'; 1 'Deactivate'

Template "Template_1" 800x480
   Button "Exit" at 722,440 size 55x39; TextOff 'Exit'; PictureOff "ExitRuntime_KTP900_Basic_PN_TR"; PictureOn "ExitRuntime_KTP900_Basic_PN_TR"
      on Release: StopRuntime(0)
   Button "Log on" at 622,440 size 55x39; TextOff 'Log on'; PictureOff "Login_KTP900_Basic_PN_TR"; PictureOn "Login_KTP900_Basic_PN_TR"
      on Release: function_a2a04561()
   Button "Template_Button" at 522,440 size 55x39; TextOff 'Text'
   Button "Template_Button_1" at 422,440 size 55x39; TextOff 'Text'
   Button "Template_Button_2" at 322,440 size 55x39; TextOff 'Text'
   Button "Template_Button_3" at 222,440 size 55x39; TextOff 'Text'
   Button "Template_Button_4" at 122,440 size 55x39; TextOff 'Text'
   Button "Start screen" at 22,440 size 55x39; TextOff 'Start screen'; PictureOff "NavigateHome_KTP900_Basic_PN_TR"; PictureOn "NavigateHome_KTP900_Basic_PN_TR"
      on Release: ActivateScreen("Root screen", 0)
   SymbolicIOField "Symbolic_IO_Field_Screen" at 74,7 size 619x26; TextOff '0'; TextOn '1'; TextList "TextList_ScreenNames"
      ProcessValue <- "Tag_ScreenNumber"
      on Change: ActivateScreenByNumber("Tag_ScreenNumber", 0)
   DateTimeField "HmiScreenItemData" at 695,20 size 105x20
   DateTimeField "HmiScreenItemData_1" at 695,0 size 105x20
   GraphicView "Logo" at 0,0 size 72x40; Picture "Logo of HMI_1"

screen "Root screen" 800x480, template "Template_1"
   on GenerateScreen: SetTag("Tag_ScreenNumber", 1)
   Circle "Circle_1" at 146,220 size 40x40
      Appearance <- "Connection_PROFINET"
   Circle "Circle_2" at 146,264 size 40x40
      Appearance <- "Connection_LOOPBACK"
   Circle "Circle_3" at 146,308 size 40x40
      Appearance <- "Connection_LOCALMODEL"
   Circle "Circle_4" at 146,176 size 40x40
      Appearance <- "Connection_NOCONNECTION"
   Circle "Circle_5" at 146,352 size 40x40
      Appearance <- "Connection_LOCALVALUE"
   Button "Button_1" at 200,220 size 110x40; TextOff 'Activate'; TextOn 'Deactivate'; TextList "Btn_ConnectionMode"
      on Click: InvertBit("Connection_PROFINET")
      ProcessValue <- "Connection_PROFINET"
   Button "Button_2" at 200,264 size 110x40; TextOn 'Deactivate'; TextOff 'Activate'; TextList "Btn_ConnectionMode"
      on Click: InvertBit("Connection_LOOPBACK")
      ProcessValue <- "Connection_LOOPBACK"
   Button "Button_3" at 200,308 size 110x40; TextOn 'Deactivate'; TextOff 'Activate'; TextList "Btn_ConnectionMode"
      on Click: InvertBit("Connection_LOCALMODEL")
      ProcessValue <- "Connection_LOCALMODEL"
   Button "Button_4" at 200,352 size 110x40; TextOn 'Deactivate'; TextOff 'Activate'; TextList "Btn_ConnectionMode"
      on Click: InvertBit("Connection_LOCALVALUE")
      ProcessValue <- "Connection_LOCALVALUE"
   TextField "Text field_1" at 110,136 size 150x25; Text 'Actual connetion'
   TextField "Text field_2" at 43,185 size 96x20; Text 'No connection'
   TextField "Text field_3" at 82,229 size 57x20; Text 'Profinet'
   TextField "Text field_4" at 73,272 size 66x20; Text 'Loopback'
   TextField "Text field_5" at 52,319 size 87x20; Text 'Local models'
   TextField "Text field_6" at 42,364 size 97x20; Text 'Manual values'
   Softkey "Softkey_F2" at 0,0 size 0x0; SoftkeyImage "Right_Arrow"
      on KeyUp: ActivateScreen("src_Regulation", 0)

screen "src_Regulation" 800x480, template "Template_1"
   TextField "Text field_7" at 508,49 size 119x25; Text 'Actual values'
   IOField "I/O field_1" at 462,74 size 96x32; FormatPattern s999999999.999
      ProcessValue <- "PID_Compact_Control_A_Input"
   IOField "I/O field_2" at 462,106 size 96x32; FormatPattern s999999999.999
      ProcessValue <- "PID_Compact_Control_B_Input"
   IOField "I/O field_3" at 462,138 size 96x32; FormatPattern s999999999.999
      ProcessValue <- "PID_Compact_Control_C_Input"
   TextField "Text field_8" at 378,80 size 56x20; Text 'PID A in'
   TextField "Text field_9" at 378,112 size 54x20; Text 'PID B in'
   TextField "Text field_10" at 378,144 size 54x20; Text 'PID C in'
   IOField "I/O field_4" at 660,74 size 96x32; FormatPattern s999999999.999
      ProcessValue <- "PID_Compact_Control_A_Output"
   IOField "I/O field_5" at 660,106 size 96x32; FormatPattern s999999999.999
      ProcessValue <- "PID_Compact_Control_B_Output"
   IOField "I/O field_6" at 660,138 size 96x32; FormatPattern s999999999.999
      ProcessValue <- "PID_Compact_Control_C_Output"
   TextField "Text field_11" at 570,80 size 67x20; Text 'PID A out'
   TextField "Text field_12" at 570,112 size 65x20; Text 'PID B out'
   TextField "Text field_13" at 570,144 size 65x20; Text 'PID C out'
   IOField "I/O field_7" at 462,179 size 96x32; FormatPattern s999999999.999
      ProcessValue <- "LSim_PDT1_DB_input"
   IOField "I/O field_8" at 462,211 size 96x32; FormatPattern s999999999.999
      ProcessValue <- "LSim_PT2aper_DB_input"
   IOField "I/O field_9" at 462,243 size 96x32; FormatPattern s999999999.999
      ProcessValue <- "LSim_PT2osc_DB_input"
   TextField "Text field_14" at 378,183 size 72x20; Text 'Model A in'
   TextField "Text field_15" at 378,215 size 70x20; Text 'Model B in'
   TextField "Text field_16" at 378,247 size 70x20; Text 'Model C in'
   IOField "I/O field_10" at 660,179 size 96x32; FormatPattern s999999999.999
      ProcessValue <- "LSim_PDT1_DB_output"
   IOField "I/O field_11" at 660,211 size 96x32; FormatPattern s999999999.999
      ProcessValue <- "LSim_PT2aper_DB_output"
   IOField "I/O field_12" at 660,243 size 96x32; FormatPattern s999999999.999
      ProcessValue <- "LSim_PT2osc_DB_output"
   TextField "Text field_17" at 570,185 size 83x20; Text 'Model A out'
   TextField "Text field_18" at 570,217 size 81x20; Text 'Model B out'
   TextField "Text field_19" at 570,249 size 81x20; Text 'Model C out'
   IOField "I/O field_13" at 462,293 size 96x32; FormatPattern s999999999.999
      ProcessValue <- "Model A - PN u"
   IOField "I/O field_14" at 462,325 size 96x32; FormatPattern s999999999.999
      ProcessValue <- "Model B - PN u"
   IOField "I/O field_15" at 462,357 size 96x32; FormatPattern s999999999.999
      ProcessValue <- "Model C - PN u"
   TextField "Text field_1" at 378,297 size 69x20; Text 'Model A u'
   TextField "Text field_2" at 378,329 size 67x20; Text 'Model B u'
   TextField "Text field_3" at 378,361 size 67x20; Text 'Model C u'
   IOField "I/O field_16" at 660,293 size 96x32; FormatPattern s999999999.999
      ProcessValue <- "Model A - PN y"
   IOField "I/O field_17" at 660,325 size 96x32; FormatPattern s999999999.999
      ProcessValue <- "Model B - PN y"
   IOField "I/O field_18" at 660,357 size 96x32; FormatPattern s999999999.999
      ProcessValue <- "Model C - PN y"
   TextField "Text field_4" at 570,299 size 69x20; Text 'Model A y'
   TextField "Text field_5" at 570,331 size 67x20; Text 'Model B y'
   TextField "Text field_6" at 570,363 size 67x20; Text 'Model C y'
   IOField "I/O field_19" at 83,262 size 87x25; FormatPattern s99.999
      ProcessValue <- "SetPoint A"
   TextField "Text field_20" at 11,266 size 60x20; Text 'Setpoint'
   IOField "I/O field_20" at 172,262 size 87x25; FormatPattern s99.999
      ProcessValue <- "SetPoint B"
   IOField "I/O field_21" at 261,262 size 87x25; FormatPattern s99.999
      ProcessValue <- "SetPoint C"
   TextField "Text field_24" at 139,49 size 102x25; Text 'Parameters'
   IOField "I/O field_22" at 83,106 size 87x25; FormatPattern s99.999
      ProcessValue <- "PID_Compact_Control_A_Retain_CtrlParams_Gain"
   TextField "Text field_25" at 10,81 size 52x20; Text 'Control'
   TextField "Text field_26" at 205,80 size 13x20; Text 'B'
   TextField "Text field_27" at 295,80 size 13x20; Text 'C'
   TextField "Text field_28" at 119,80 size 15x20; Text 'A'
   TextField "Text field_29" at 20,110 size 32x20; Text 'Gain'
   TextField "Text field_30" at 27,140 size 15x20; Text 'Ti'
   TextField "Text field_31" at 25,171 size 20x20; Text 'Td'
   IOField "I/O field_23" at 83,137 size 87x25; FormatPattern s99.999
      ProcessValue <- "PID_Compact_Control_A_Retain_CtrlParams_Ti"
   IOField "I/O field_24" at 83,167 size 87x25; FormatPattern s99.999
      ProcessValue <- "PID_Compact_Control_A_Retain_CtrlParams_Td"
   IOField "I/O field_25" at 172,106 size 87x25; FormatPattern s99.999
      ProcessValue <- "PID_Compact_Control_B_Retain_CtrlParams_Gain"
   IOField "I/O field_26" at 172,137 size 87x25; FormatPattern s99.999
      ProcessValue <- "PID_Compact_Control_B_Retain_CtrlParams_Ti"
   IOField "I/O field_27" at 172,167 size 87x25; FormatPattern s99.999
      ProcessValue <- "PID_Compact_Control_B_Retain_CtrlParams_Td"
   IOField "I/O field_28" at 261,106 size 87x25; FormatPattern s99.999
      ProcessValue <- "PID_Compact_Control_C_Retain_CtrlParams_Gain"
   IOField "I/O field_29" at 261,137 size 87x25; FormatPattern s99.999
      ProcessValue <- "PID_Compact_Control_C_Retain_CtrlParams_Ti"
   IOField "I/O field_30" at 261,167 size 87x25; FormatPattern s99.999
      ProcessValue <- "PID_Compact_Control_C_Retain_CtrlParams_Td"
   TextField "Text field_32" at 18,201 size 39x20; Text 'Cycle'
   IOField "I/O field_31" at 83,197 size 87x25; FormatPattern s99.999
      ProcessValue <- "PID_Compact_Control_A_Retain_CtrlParams_Cycle"
   IOField "I/O field_32" at 172,197 size 87x25; FormatPattern s99.999
      ProcessValue <- "PID_Compact_Control_B_Retain_CtrlParams_Cycle"
   IOField "I/O field_33" at 261,197 size 87x25; FormatPattern s99.999
      ProcessValue <- "PID_Compact_Control_C_Retain_CtrlParams_Cycle"
   TextField "Text field_21" at 539,275 size 64x20; Text 'PROFINET'
   TextField "Text field_22" at 142,297 size 75x25; Text 'Model D'
   TextField "Text field_23" at 18,355 size 60x20; Text 'Setpoint'
   TextField "Text field_33" at 185,328 size 32x20; Text 'Gain'
   TextField "Text field_34" at 202,355 size 15x20; Text 'Ti'
   TextField "Text field_35" at 198,383 size 20x20; Text 'Td'
   TextField "Text field_36" at 28,330 size 39x20; Text 'Cycle'
   IOField "I/O field_34" at 85,353 size 87x25; FormatPattern s99.999
      ProcessValue <- "SetPoint D"
   IOField "I/O field_35" at 85,328 size 87x25; FormatPattern s99.999
      ProcessValue <- "PID_Compact_Control_D_Retain_CtrlParams_Cycle"
   IOField "I/O field_36" at 232,378 size 87x25; FormatPattern s99.999
      ProcessValue <- "PID_Compact_Control_D_Retain_CtrlParams_Td"
   IOField "I/O field_37" at 232,353 size 87x25; FormatPattern s99.999
      ProcessValue <- "PID_Compact_Control_D_Retain_CtrlParams_Ti"
   IOField "I/O field_38" at 232,328 size 87x25; FormatPattern s99.999
      ProcessValue <- "PID_Compact_Control_D_Retain_CtrlParams_Gain"
   IOField "I/O field_39" at 462,389 size 96x32; FormatPattern s999999999.999
      ProcessValue <- "Model D - PN u"
   IOField "I/O field_40" at 660,389 size 96x32; FormatPattern s999999999.999
      ProcessValue <- "Model D - PN y"
   TextField "Text field_37" at 570,395 size 68x20; Text 'Model D y'
   TextField "Text field_38" at 378,394 size 68x20; Text 'Model D u'
*)